// Mitsubishi GX Works2 project: BookEX6_1 Lib   PLC: Q13UDV

// global labels: Global
VAR_GLOBAL
  bVar0 AT M5000 : BOOL;
  abArray0 AT M5010 : ARRAY [0..49] OF BOOL;
  sStr0 AT D5000 : STRING[199];
  sStr1 AT D5100 : STRING[199];
  sStr2 AT D5200 : STRING[199];
  sStr3 AT D5300 : STRING[199];
  sStr4 AT D5400 : STRING[199];
  sStr5 AT D5500 : STRING[199];
  sStr6 AT D5600 : STRING[199];
  sStr7 AT D5700 : STRING[199];
  sStr8 AT D5800 : STRING[199];
  sStr9 AT D5900 : STRING[199];
  iVar0 AT D4500 : INT;
  iVar1 AT D4501 : INT;
  iVar2 AT D4502 : INT;
  iVar3 AT D4503 : INT;
  iVar4 AT D4504 : INT;
  iVar5 AT D4505 : INT;
  iVar6 AT D4506 : INT;
  iVar7 AT D4507 : INT;
  iVar8 AT D4508 : INT;
  iVar9 AT D4509 : INT;
  dVar0 AT D4510 : DINT;
  dVar1 AT D4512 : DINT;
  dVar2 AT D4514 : DINT;
  dVar3 AT D4516 : DINT;
  dVar4 AT D4518 : DINT;
  dVar5 AT D4520 : DINT;
  dVar6 AT D4522 : DINT;
  dVar7 AT D4524 : DINT;
  dVar8 AT D4526 : DINT;
  dVar9 AT D4528 : DINT;
  wVar0 AT D4530 : WORD;
  wVar1 AT D4531 : WORD;
  wVar2 AT D4532 : WORD;
  wVar3 AT D4533 : WORD;
  wVar4 AT D4534 : WORD;
  wVar5 AT D4535 : WORD;
  wVar6 AT D4536 : WORD;
  wVar7 AT D4537 : WORD;
  wVar8 AT D4538 : WORD;
  wVar9 AT D4539 : WORD;
  dwVar0 AT D4540 : DWORD;
  dwVar1 AT D4542 : DWORD;
  dwVar2 AT D4544 : DWORD;
  dwVar3 AT D4546 : DWORD;
  dwVar4 AT D4548 : DWORD;
  dwVar5 AT D4550 : DWORD;
  dwVar6 AT D4552 : DWORD;
  dwVar7 AT D4554 : DWORD;
  dwVar8 AT D4556 : DWORD;
  dwVar9 AT D4558 : DWORD;
  fsVar0 AT D4560 : REAL;
  fsVar1 AT D4562 : REAL;
  fsVar2 AT D4564 : REAL;
  fsVar3 AT D4566 : REAL;
  fsVar4 AT D4568 : REAL;
  fsVar5 AT D4570 : REAL;
  fsVar6 AT D4572 : REAL;
  fsVar7 AT D4574 : REAL;
  fsVar8 AT D4576 : REAL;
  fsVar9 AT D4578 : REAL;
  fdVar0 AT D4580 : LREAL;
  tTime0 AT D4620 : TIME;
  tTime1 AT D4622 : TIME;
  tTime2 AT D4624 : TIME;
  tTime3 AT D4626 : TIME;
  tTime4 AT D4628 : TIME;
  tTime5 AT D4630 : TIME;
  tTime6 AT D4632 : TIME;
  tTime7 AT D4634 : TIME;
  tTime8 AT D4636 : TIME;
  tTime9 AT D4638 : TIME;
  tTime10 AT D4640 : TIME;
  bVar1 AT M5001 : BOOL;
  bVar2 AT M5002 : BOOL;
  bVar3 AT M5003 : BOOL;
  bVar4 AT M5004 : BOOL;
  bVar5 AT M5005 : BOOL;
  bVar6 AT M5006 : BOOL;
  bVar7 AT M5007 : BOOL;
  bVar8 AT M5008 : BOOL;
  bVar9 AT M5009 : BOOL;
  abArray1 AT M5060 : ARRAY [0..49] OF BOOL;
  abArray2 AT M5110 : ARRAY [0..49] OF BOOL;
  abArray3 AT M5160 : ARRAY [0..49] OF BOOL;
  abArray4 AT M5210 : ARRAY [0..49] OF BOOL;
  abArray5 AT M5260 : ARRAY [0..49] OF BOOL;
  abArray6 AT M5310 : ARRAY [0..49] OF BOOL;
  abArray7 AT M5360 : ARRAY [0..49] OF BOOL;
  abArray8 AT M5410 : ARRAY [0..49] OF BOOL;
  abArray9 AT M5460 : ARRAY [0..49] OF BOOL;
  fdVar1 AT D4584 : LREAL;
  fdVar2 AT D4588 : LREAL;
  fdVar3 AT D4592 : LREAL;
  fdVar4 AT D4596 : LREAL;
  fdVar5 AT D4600 : LREAL;
  fdVar6 AT D4604 : LREAL;
  fdVar7 AT D4608 : LREAL;
  fdVar8 AT D4612 : LREAL;
  fdVar9 AT D4616 : LREAL;
  afsPen0 AT D2000 : ARRAY [0..499] OF REAL;
  afsPen1 AT D3000 : ARRAY [0..499] OF REAL;
  adwD10 AT D10 : ARRAY [0..9] OF DWORD;
  awD10 AT D10 : ARRAY [0..19] OF WORD;
  abM10 AT M10 : ARRAY [0..19] OF BOOL;
END_VAR
// user libraries (not included): HMI

PROGRAM ExEtc
VAR
  HMI05_1 : HMI05;
  bSendOK : BOOL;
  abCloseComp : ARRAY [0..1] OF BOOL;
  bSendErr : BOOL;
END_VAR
(* structured ladder/FBD written out as ST: instructions are called as NAME(EN, inputs, outputs); _pN, _eN, _tN stand for wires *)
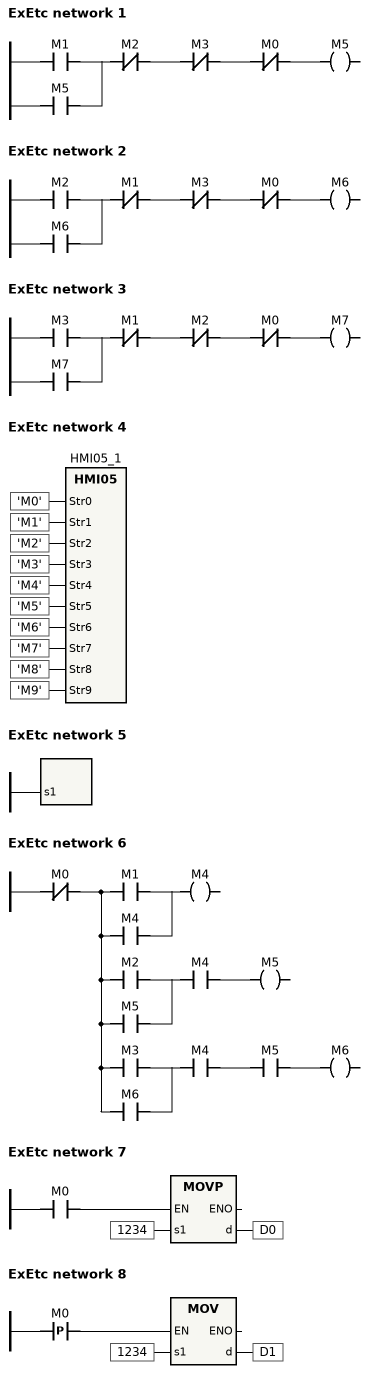
(* network 1 *)
M5 := (((M1 OR M5) AND NOT M2) AND NOT M3) AND NOT M0;
(* network 2 *)
M6 := (((M2 OR M6) AND NOT M1) AND NOT M3) AND NOT M0;
(* network 3 *)
M7 := (((M3 OR M7) AND NOT M1) AND NOT M2) AND NOT M0;
(* network 4 *)
HMI05_1(Str0 := 'M0', Str1 := 'M1', Str2 := 'M2', Str3 := 'M3', Str4 := 'M4', Str5 := 'M5', Str6 := 'M6', Str7 := 'M7', Str8 := 'M8', Str9 := 'M9');
(* network 5 *)
(* element kind 10  <- TRUE *)
(* network 6 *)
_p1 := NOT M0;
M4 := (_p1 AND M1) OR (_p1 AND M4);
M5 := ((_p1 AND M2) OR (_p1 AND M5)) AND M4;
M6 := (((_p1 AND M3) OR (_p1 AND M6)) AND M4) AND M5;
(* network 7 *)
MOVP(M0, 1234, D0);
(* network 8 *)
MOV(LDP(TRUE, M0), 1234, D1);
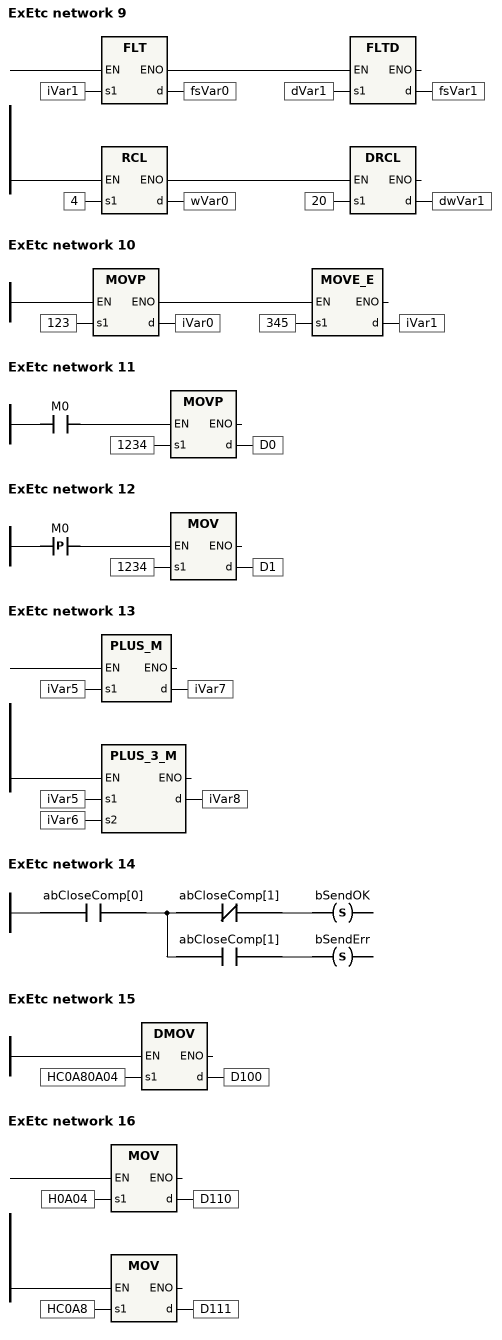
(* network 9 *)
_e1 := FLT(TRUE, iVar1, fsVar0);
FLTD(_e1, dVar1, fsVar1);
_e2 := RCL(TRUE, 4, wVar0);
DRCL(_e2, 20, dwVar1);
(* network 10 *)
_e1 := MOVP(TRUE, 123, iVar0);
MOVE_E(_e1, 345, iVar1);
(* network 11 *)
MOVP(M0, 1234, D0);
(* network 12 *)
MOV(LDP(TRUE, M0), 1234, D1);
(* network 13 *)
PLUS_M(TRUE, iVar5, iVar7);
PLUS_3_M(TRUE, iVar5, iVar6, iVar8);
(* network 14 *)
SET(abCloseComp[0] AND NOT abCloseComp[1], bSendOK);
SET(abCloseComp[0] AND abCloseComp[1], bSendErr);
(* network 15 *)
DMOV(TRUE, HC0A80A04, D100);
(* network 16 *)
MOV(TRUE, H0A04, D110);
MOV(TRUE, HC0A8, D111);
END_PROGRAM

PROGRAM ExMovBit
VAR
  Mov4BIT_1 : Mov4BIT;
  Mov8BIT_1 : Mov8BIT;
END_VAR
(* structured ladder/FBD written out as ST: instructions are called as NAME(EN, inputs, outputs); _pN, _eN, _tN stand for wires *)
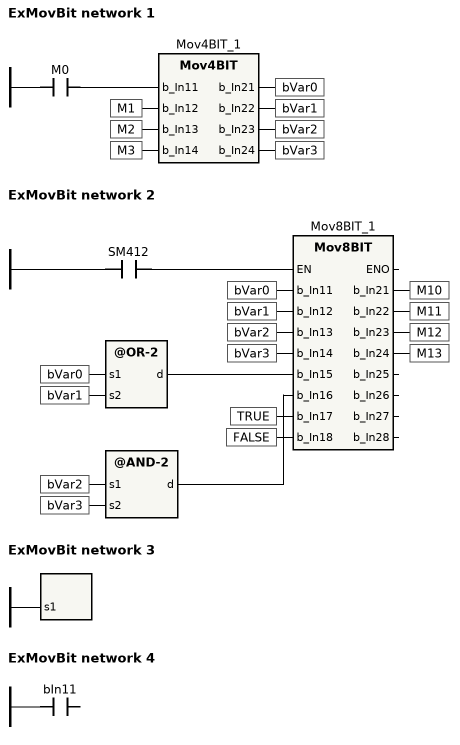
(* network 1 *)
Mov4BIT_1(b_In11 := M0, b_In12 := M1, b_In13 := M2, b_In14 := M3, b_In21 => bVar0, b_In22 => bVar1, b_In23 => bVar2, b_In24 => bVar3);
(* network 2 *)
Mov8BIT_1(EN := SM412, b_In11 := bVar0, b_In12 := bVar1, b_In13 := bVar2, b_In14 := bVar3, b_In15 := @OR-2(bVar0, bVar1), b_In16 := @AND-2(bVar2, bVar3), b_In17 := TRUE, b_In18 := FALSE, b_In21 => M10, b_In22 => M11, b_In23 => M12, b_In24 => M13);
(* network 3 *)
(* element kind 10  <- TRUE *)
(* network 4 *)
(* not connected to any output: bIn11 *)
END_PROGRAM

PROGRAM ExMovINT
VAR
  Mov4INT_1 : Mov4INT;
  Mov8INT_1 : Mov8INT;
  Mov4INT_2 : Mov4INT;
  Mov4INT_3 : Mov4INT;
END_VAR
(* structured ladder/FBD written out as ST: instructions are called as NAME(EN, inputs, outputs); _pN, _eN, _tN stand for wires *)
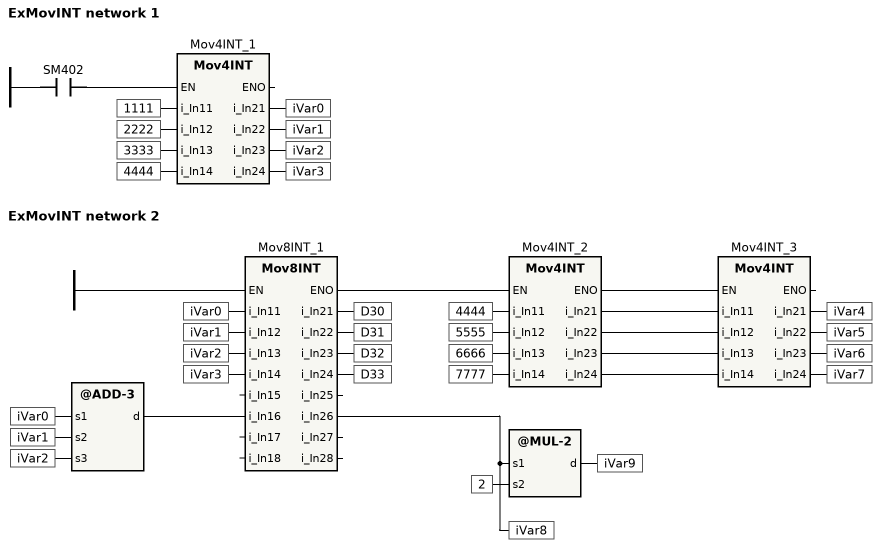
(* network 1 *)
Mov4INT_1(EN := SM402, i_In11 := 1111, i_In12 := 2222, i_In13 := 3333, i_In14 := 4444, i_In21 => iVar0, i_In22 => iVar1, i_In23 => iVar2, i_In24 => iVar3);
(* network 2 *)
Mov8INT_1(EN := TRUE, i_In11 := iVar0, i_In12 := iVar1, i_In13 := iVar2, i_In14 := iVar3, i_In16 := @ADD-3(iVar0, iVar1, iVar2), i_In21 => D30, i_In22 => D31, i_In23 => D32, i_In24 => D33);
Mov4INT_2(EN := Mov8INT_1.ENO, i_In11 := 4444, i_In12 := 5555, i_In13 := 6666, i_In14 := 7777);
Mov4INT_3(EN := Mov4INT_2.ENO, i_In11 := Mov4INT_2.i_In21, i_In12 := Mov4INT_2.i_In22, i_In13 := Mov4INT_2.i_In23, i_In14 := Mov4INT_2.i_In24, i_In21 => iVar4, i_In22 => iVar5, i_In23 => iVar6, i_In24 => iVar7);
iVar9 := @MUL-2(Mov8INT_1.i_In26, 2);
iVar8 := Mov8INT_1.i_In26;
END_PROGRAM

PROGRAM ExMovWORD
VAR
  Mov4WORD_1 : Mov4WORD;
  Mov8WORD_1 : Mov8WORD;
  Mov4WORD_2 : Mov4WORD;
END_VAR
(* structured ladder/FBD written out as ST: instructions are called as NAME(EN, inputs, outputs); _pN, _eN, _tN stand for wires *)
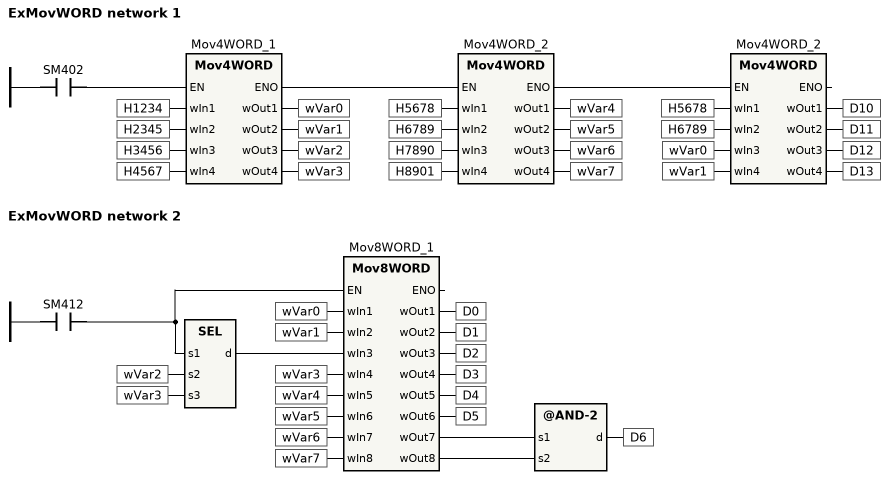
(* network 1 *)
Mov4WORD_1(EN := SM402, wIn1 := H1234, wIn2 := H2345, wIn3 := H3456, wIn4 := H4567, wOut1 => wVar0, wOut2 => wVar1, wOut3 => wVar2, wOut4 => wVar3);
Mov4WORD_2(EN := Mov4WORD_1.ENO, wIn1 := H5678, wIn2 := H6789, wIn3 := H7890, wIn4 := H8901, wOut1 => wVar4, wOut2 => wVar5, wOut3 => wVar6, wOut4 => wVar7);
Mov4WORD_2(EN := Mov4WORD_2.ENO, wIn1 := H5678, wIn2 := H6789, wIn3 := wVar0, wIn4 := wVar1, wOut1 => D10, wOut2 => D11, wOut3 => D12, wOut4 => D13);
(* network 2 *)
Mov8WORD_1(EN := SM412, wIn1 := wVar0, wIn2 := wVar1, wIn3 := SEL(SM412, wVar2, wVar3), wIn4 := wVar3, wIn5 := wVar4, wIn6 := wVar5, wIn7 := wVar6, wIn8 := wVar7, wOut1 => D0, wOut2 => D1, wOut3 => D2, wOut4 => D3, wOut5 => D4, wOut6 => D5);
D6 := @AND-2(Mov8WORD_1.wOut7, Mov8WORD_1.wOut8);
END_PROGRAM

PROGRAM ExMovREAL
VAR
  Mov4REAL_1 : Mov4REAL;
  Mov8REAL_1 : Mov8REAL;
END_VAR
(* structured ladder/FBD written out as ST: instructions are called as NAME(EN, inputs, outputs); _pN, _eN, _tN stand for wires *)
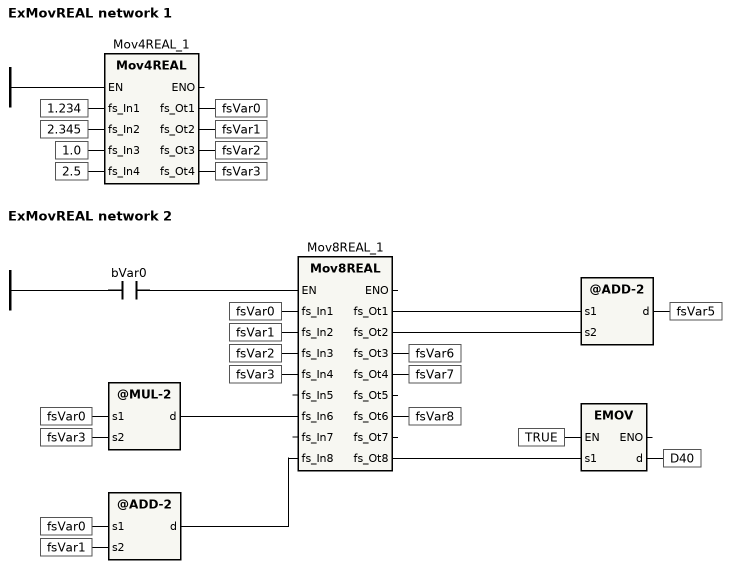
(* network 1 *)
Mov4REAL_1(EN := TRUE, fs_In1 := 1.234, fs_In2 := 2.345, fs_In3 := 1.0, fs_In4 := 2.5, fs_Ot1 => fsVar0, fs_Ot2 => fsVar1, fs_Ot3 => fsVar2, fs_Ot4 => fsVar3);
(* network 2 *)
Mov8REAL_1(EN := bVar0, fs_In1 := fsVar0, fs_In2 := fsVar1, fs_In3 := fsVar2, fs_In4 := fsVar3, fs_In6 := @MUL-2(fsVar0, fsVar3), fs_In8 := @ADD-2(fsVar0, fsVar1), fs_Ot3 => fsVar6, fs_Ot4 => fsVar7, fs_Ot6 => fsVar8);
fsVar5 := @ADD-2(Mov8REAL_1.fs_Ot1, Mov8REAL_1.fs_Ot2);
EMOV(TRUE, Mov8REAL_1.fs_Ot8, D40);
END_PROGRAM

PROGRAM ExHMI01
VAR
  HMI01_1 : HMI01;
  HMI01_2 : HMI01;
END_VAR
(* structured ladder/FBD written out as ST: instructions are called as NAME(EN, inputs, outputs); _pN, _eN, _tN stand for wires *)
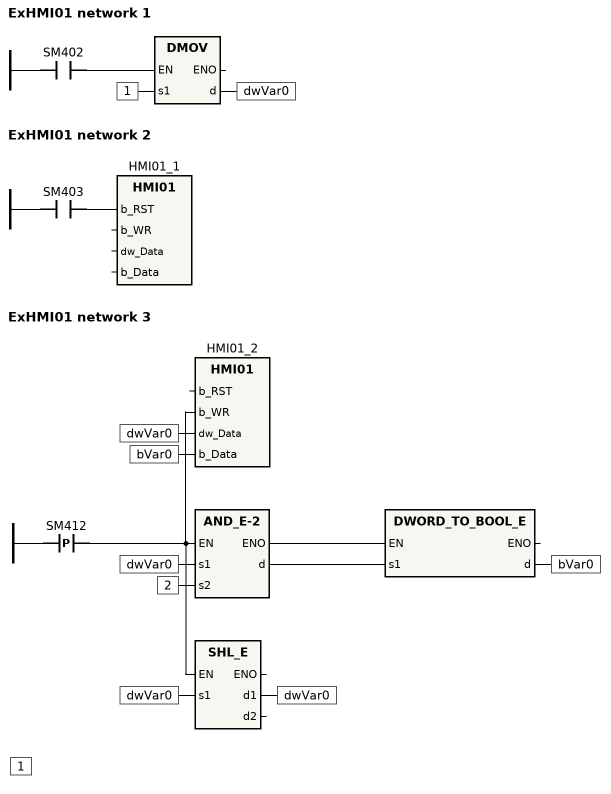
(* network 1 *)
DMOV(SM402, 1, dwVar0);
(* network 2 *)
HMI01_1(b_RST := SM403);
(* network 3 *)
_p1 := LDP(TRUE, SM412);
HMI01_2(b_WR := _p1, dw_Data := dwVar0, b_Data := bVar0);
SHL_E(_p1, dwVar0, dwVar0, _open);
_e3 := AND_E(_p1, dwVar0, 2, _t2);
DWORD_TO_BOOL_E(_e3, _t2, bVar0);
(* not connected to any output: 1 *)
END_PROGRAM

PROGRAM ExHMI02
VAR
  HMI02_1 : HMI02;
  TON_1 : TON;
  TON_2 : TON;
END_VAR
(* structured ladder/FBD written out as ST: instructions are called as NAME(EN, inputs, outputs); _pN, _eN, _tN stand for wires *)
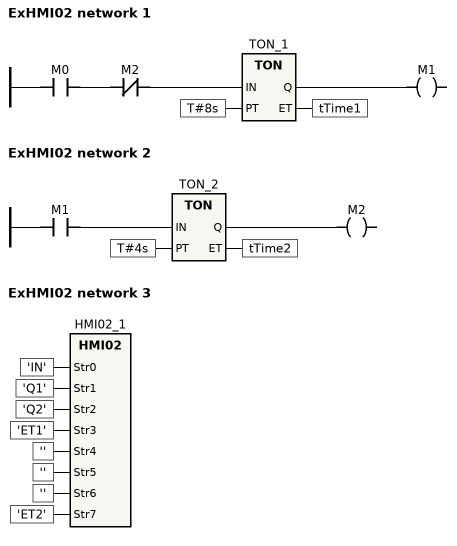
(* network 1 *)
TON_1(IN := M0 AND NOT M2, PT := T#8s, ET => tTime1);
M1 := TON_1.Q;
(* network 2 *)
TON_2(IN := M1, PT := T#4s, ET => tTime2);
M2 := TON_2.Q;
(* network 3 *)
HMI02_1(Str0 := 'IN', Str1 := 'Q1', Str2 := 'Q2', Str3 := 'ET1', Str4 := '', Str5 := '', Str6 := '', Str7 := 'ET2');
END_PROGRAM

PROGRAM ExHMI03
VAR
  HMI03_1 : HMI03;
  TON_E_1 : TON_E;
END_VAR
(* structured ladder/FBD written out as ST: instructions are called as NAME(EN, inputs, outputs); _pN, _eN, _tN stand for wires *)
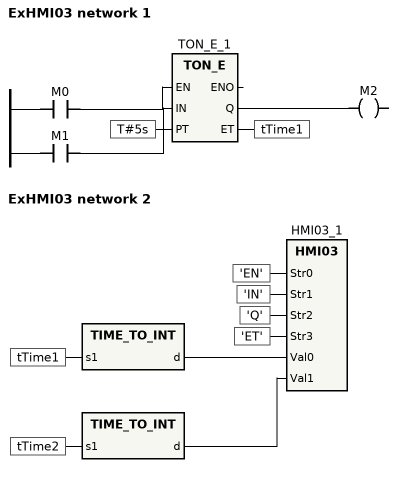
(* network 1 *)
TON_E_1(EN := M0, IN := M1, PT := T#5s, ET => tTime1);
M2 := TON_E_1.Q;
(* network 2 *)
HMI03_1(Str0 := 'EN', Str1 := 'IN', Str2 := 'Q', Str3 := 'ET', Val0 := TIME_TO_INT(tTime1), Val1 := TIME_TO_INT(tTime2));
END_PROGRAM

PROGRAM ExHMI04
VAR
  HMI04_1 : HMI04;
  TON_E_1 : TON_E;
  TON_E_2 : TON_E;
END_VAR
(* structured ladder/FBD written out as ST: instructions are called as NAME(EN, inputs, outputs); _pN, _eN, _tN stand for wires *)
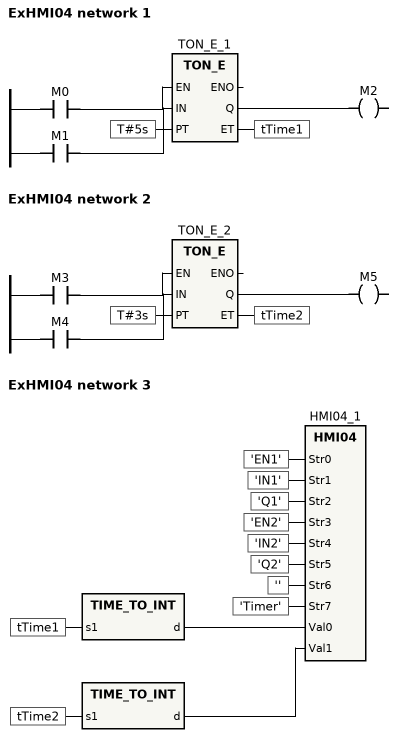
(* network 1 *)
TON_E_1(EN := M0, IN := M1, PT := T#5s, ET => tTime1);
M2 := TON_E_1.Q;
(* network 2 *)
TON_E_2(EN := M3, IN := M4, PT := T#3s, ET => tTime2);
M5 := TON_E_2.Q;
(* network 3 *)
HMI04_1(Str0 := 'EN1', Str1 := 'IN1', Str2 := 'Q1', Str3 := 'EN2', Str4 := 'IN2', Str5 := 'Q2', Str6 := '', Str7 := 'Timer', Val0 := TIME_TO_INT(tTime1), Val1 := TIME_TO_INT(tTime2));
END_PROGRAM

PROGRAM ExHMI05
VAR
  HMI05_1 : HMI05;
END_VAR
(* structured ladder/FBD written out as ST: instructions are called as NAME(EN, inputs, outputs); _pN, _eN, _tN stand for wires *)
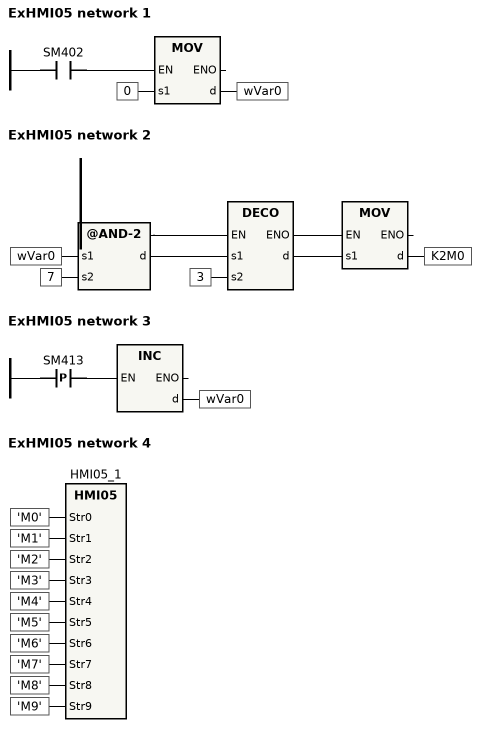
(* network 1 *)
MOV(SM402, 0, wVar0);
(* network 2 *)
_e2 := DECO(TRUE, @AND-2(wVar0, 7), 3, _t1);
MOV(_e2, _t1, K2M0);
(* network 3 *)
INC(LDP(TRUE, SM413), wVar0);
(* network 4 *)
HMI05_1(Str0 := 'M0', Str1 := 'M1', Str2 := 'M2', Str3 := 'M3', Str4 := 'M4', Str5 := 'M5', Str6 := 'M6', Str7 := 'M7', Str8 := 'M8', Str9 := 'M9');
END_PROGRAM

PROGRAM ExHMI06
VAR
  HMI06_1 : HMI06;
  ix : INT;
  iy : INT;
  radx : REAL;
  fsx1 : REAL;
  fsx2 : REAL;
  fscale : REAL;
END_VAR
(* structured ladder/FBD written out as ST: instructions are called as NAME(EN, inputs, outputs); _pN, _eN, _tN stand for wires *)
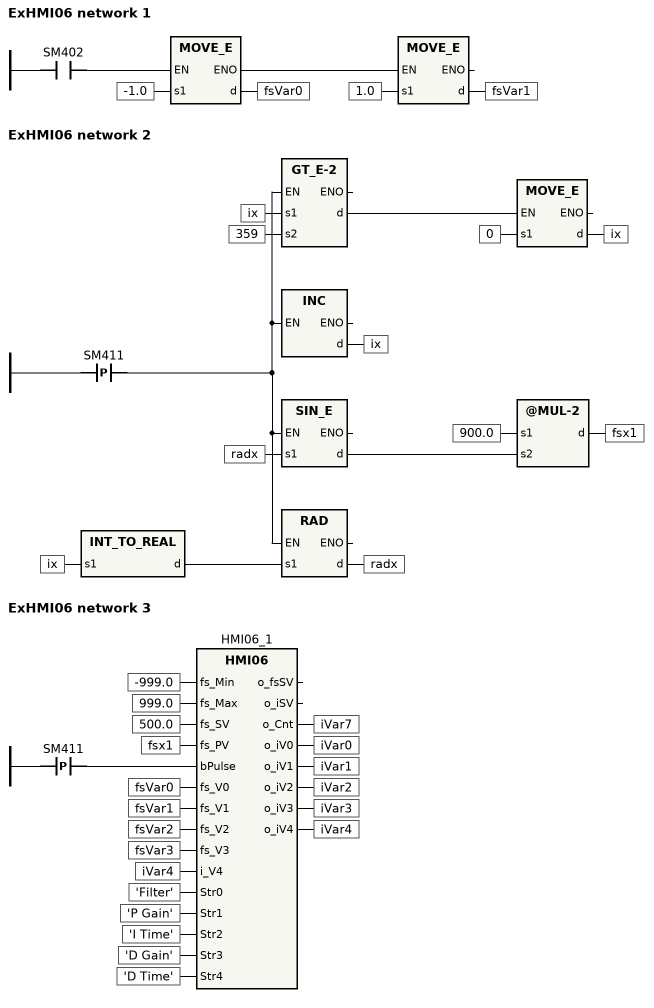
(* network 1 *)
_e1 := MOVE_E(SM402, -1.0, fsVar0);
MOVE_E(_e1, 1.0, fsVar1);
(* network 2 *)
_p1 := LDP(TRUE, SM411);
INC(_p1, ix);
GT_E(_p1, ix, 359, _t2);
MOVE_E(_t2, 0, ix);
RAD(_p1, INT_TO_REAL(ix), radx);
SIN_E(_p1, radx, _t3);
fsx1 := @MUL-2(900.0, _t3);
(* network 3 *)
HMI06_1(fs_Min := -999.0, fs_Max := 999.0, fs_SV := 500.0, fs_PV := fsx1, bPulse := LDP(TRUE, SM411), fs_V0 := fsVar0, fs_V1 := fsVar1, fs_V2 := fsVar2, fs_V3 := fsVar3, i_V4 := iVar4, Str0 := 'Filter', Str1 := 'P Gain', Str2 := 'I Time', Str3 := 'D Gain', Str4 := 'D Time', o_Cnt => iVar7, o_iV0 => iVar0, o_iV1 => iVar1, o_iV2 => iVar2, o_iV3 => iVar3, o_iV4 => iVar4);
END_PROGRAM

PROGRAM ExHMI20
VAR
  HMI20_1 : HMI20;
END_VAR
(* structured ladder/FBD written out as ST: instructions are called as NAME(EN, inputs, outputs); _pN, _eN, _tN stand for wires *)
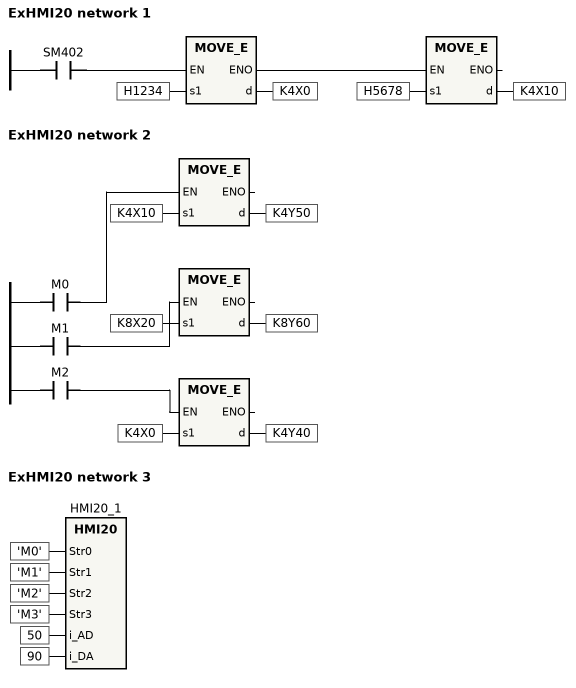
(* network 1 *)
_e1 := MOVE_E(SM402, H1234, K4X0);
MOVE_E(_e1, H5678, K4X10);
(* network 2 *)
MOVE_E(M0, K4X10, K4Y50);
MOVE_E(M1, K8X20, K8Y60);
MOVE_E(M2, K4X0, K4Y40);
(* network 3 *)
HMI20_1(Str0 := 'M0', Str1 := 'M1', Str2 := 'M2', Str3 := 'M3', i_AD := 50, i_DA := 90);
END_PROGRAM

PROGRAM ExMovDWORD
VAR
  Mov4DWORD_1 : Mov4DWORD;
  Mov8DWORD_1 : Mov8DWORD;
  Mov4DWORD_2 : Mov4DWORD;
END_VAR
(* structured ladder/FBD written out as ST: instructions are called as NAME(EN, inputs, outputs); _pN, _eN, _tN stand for wires *)
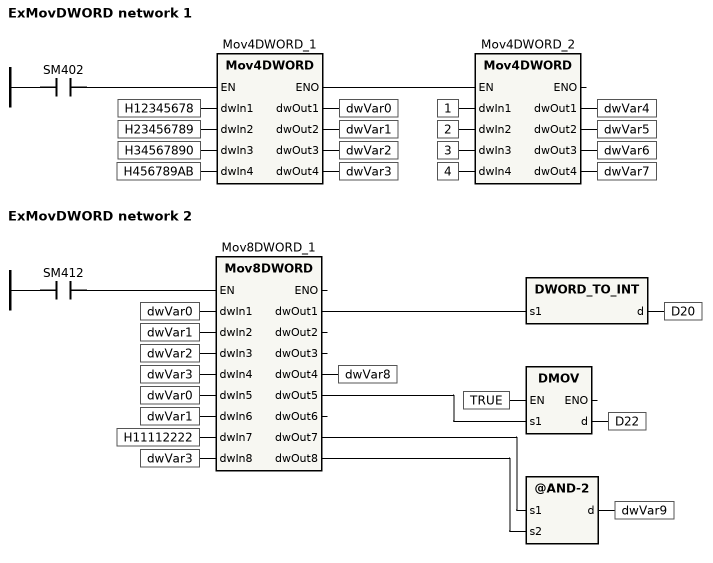
(* network 1 *)
Mov4DWORD_1(EN := SM402, dwIn1 := H12345678, dwIn2 := H23456789, dwIn3 := H34567890, dwIn4 := H456789AB, dwOut1 => dwVar0, dwOut2 => dwVar1, dwOut3 => dwVar2, dwOut4 => dwVar3);
Mov4DWORD_2(EN := Mov4DWORD_1.ENO, dwIn1 := 1, dwIn2 := 2, dwIn3 := 3, dwIn4 := 4, dwOut1 => dwVar4, dwOut2 => dwVar5, dwOut3 => dwVar6, dwOut4 => dwVar7);
(* network 2 *)
Mov8DWORD_1(EN := SM412, dwIn1 := dwVar0, dwIn2 := dwVar1, dwIn3 := dwVar2, dwIn4 := dwVar3, dwIn5 := dwVar0, dwIn6 := dwVar1, dwIn7 := H11112222, dwIn8 := dwVar3, dwOut4 => dwVar8);
D20 := DWORD_TO_INT(Mov8DWORD_1.dwOut1);
DMOV(TRUE, Mov8DWORD_1.dwOut5, D22);
dwVar9 := @AND-2(Mov8DWORD_1.dwOut7, Mov8DWORD_1.dwOut8);
END_PROGRAM

PROGRAM ExHMI08_ST
VAR
  ix : INT;
  radx : REAL;
  fsx1 : REAL;
  fsx2 : REAL;
  fscale : REAL;
  HMI08_1 : HMI08;
  iy : INT;
END_VAR
 
IF SM402 THEN
	fsVar8 := -1.0;		 (* MIN Y *)
	fsVar9 := 1.0;		 (* MAX Y *)	
END_IF;
IF LDP(TRUE, SM411) THEN 
	ix := ix + 1; 
	IF ix > 359 THEN ix := 0; END_IF;
	RAD(TRUE,INT_TO_REAL(ix),radx);
	SIN_E(TRUE, radx, fsx1);
	COS_E(TRUE, radx, fsx2);
	HMI08_1(EN:= TRUE, fs_D0:= fsx1, fs_D1:= fsx2, fs_min:= fsVar8, fs_max:= fsVar9);
	iVar7 := HMI08_1.o_min;
	iVar8 := HMI08_1.o_mid;
	iVar9 := HMI08_1.o_max;
END_IF;
END_PROGRAM

PROGRAM ExHMI08_LD
VAR
  ix : INT;
  iy : INT;
  radx : REAL;
  fsx1 : REAL;
  fsx2 : REAL;
  fscale : REAL;
  HMI08_1 : HMI08;
END_VAR
(* structured ladder/FBD written out as ST: instructions are called as NAME(EN, inputs, outputs); _pN, _eN, _tN stand for wires *)
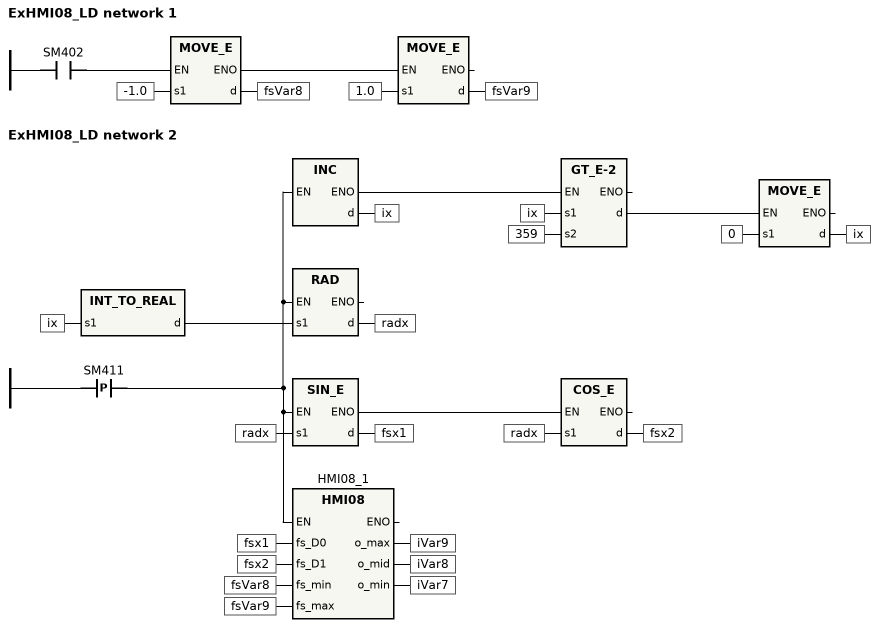
(* network 1 *)
_e1 := MOVE_E(SM402, -1.0, fsVar8);
MOVE_E(_e1, 1.0, fsVar9);
(* network 2 *)
_p1 := LDP(TRUE, SM411);
_e2 := INC(_p1, ix);
GT_E(_e2, ix, 359, _t3);
MOVE_E(_t3, 0, ix);
RAD(_p1, INT_TO_REAL(ix), radx);
_e4 := SIN_E(_p1, radx, fsx1);
COS_E(_e4, radx, fsx2);
HMI08_1(EN := _p1, fs_D0 := fsx1, fs_D1 := fsx2, fs_min := fsVar8, fs_max := fsVar9, o_max => iVar9, o_mid => iVar8, o_min => iVar7);
END_PROGRAM

PROGRAM ExHMI15
VAR
  CTU_E_1 : CTU_E;
  HMI15_1 : HMI15;
END_VAR
(* structured ladder/FBD written out as ST: instructions are called as NAME(EN, inputs, outputs); _pN, _eN, _tN stand for wires *)
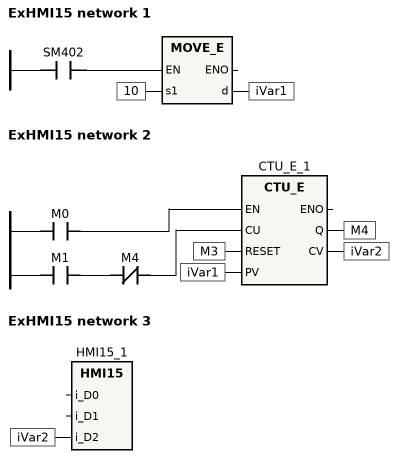
(* network 1 *)
MOVE_E(SM402, 10, iVar1);
(* network 2 *)
CTU_E_1(EN := M0, CU := M1 AND NOT M4, RESET := M3, PV := iVar1, Q => M4, CV => iVar2);
(* network 3 *)
HMI15_1(i_D2 := iVar2);
END_PROGRAM
